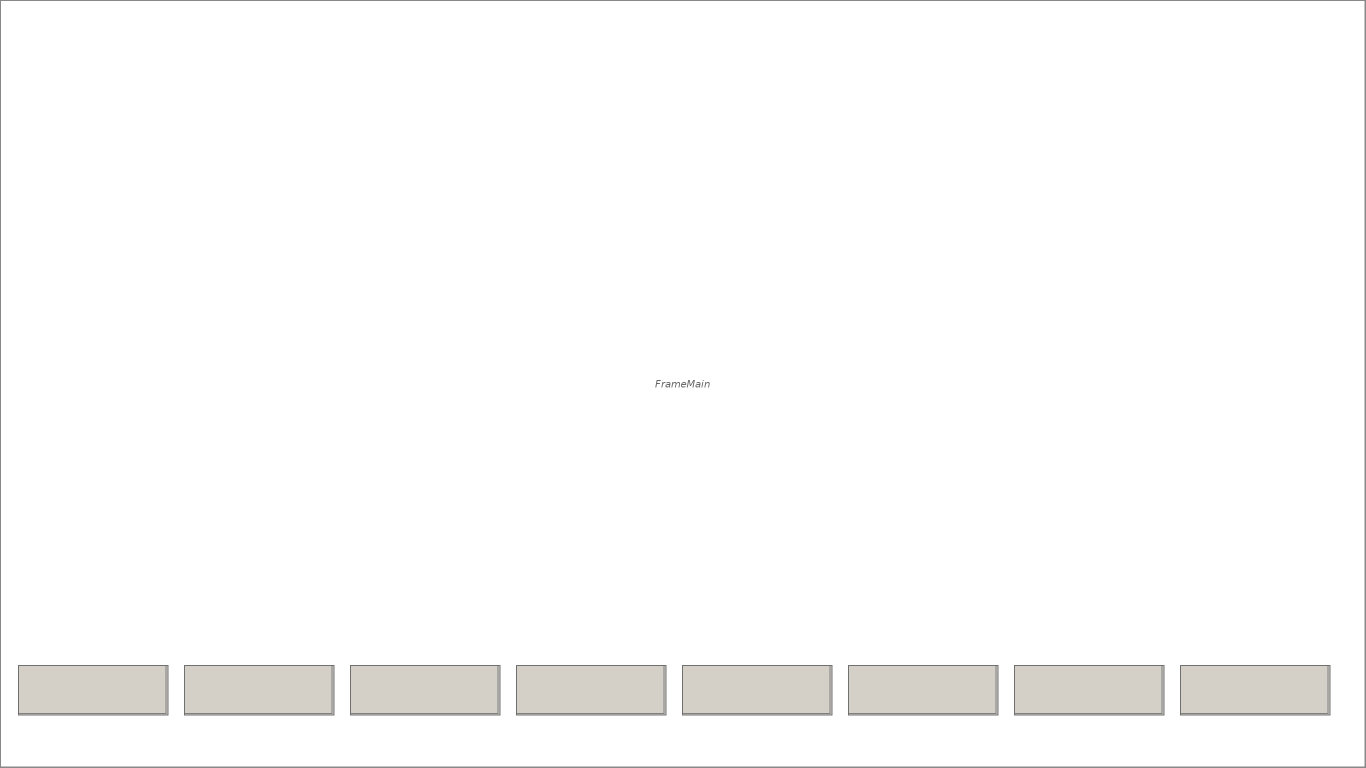
VISUALIZATION CtrlPageSetting  // 1366x768
    Frame (0,0 1366x768)
        shows FrameMain()
    Button (18,665 150x50), text list: 'StationName', text index: 0
        OnMouseClick: change screen: PageSetting_AcquireLoad
    Button (184,665 150x50), text list: 'StationName', text index: 1
        OnMouseClick: change screen: PageSetting_Steering
    Button (350,665 150x50), text list: 'StationName', text index: 2
        OnMouseClick: change screen: PageSetting_OpenLock
    Button (516,665 150x50), text list: 'StationName', text index: 3
        OnMouseClick: change screen: PageSetting_TakeUc
    Button (682,665 150x50), text list: 'StationName', text index: 4
        OnMouseClick: change screen: PageSetting_TakeUc_M
    Button (848,665 150x50), text list: 'StationName', text index: 5
        OnMouseClick: change screen: PageSetting_UnloadFrock
    Button (1014,665 150x50), text list: 'StationName', text index: 6
        OnMouseClick: change screen: PageSetting_Unload_L
    Button (1180,665 150x50), text list: 'StationName', text index: 7
        OnMouseClick: change screen: PageSetting_Other
END_VISUALIZATION

(* stored: Version 1.1.0.1, ProductVersion 3.1.4024.3
   Visu CtrlPageSetting: Id {d6252887-db92-4583-8fb1-33e7bb357cb8} *)
